Staubli VAL3: MoveTo.pgx

program MoveTo(pointRx x_pPoint, tool x_tTool, mdesc x_mDesc, num x_nMoveType, bool& x_bUnReachable)
  local string l_sMessage
  local joint l_jJoint
begin
  if pointToJoint(x_tTool,herej(),x_pPoint,l_jJoint)
    switch x_nMoveType
      case 0
        movel(x_pPoint,x_tTool,x_mDesc)
      break
      case 1
        movej(x_pPoint,x_tTool,x_mDesc)
      break
    endSwitch
  else
     x_bUnReachable=true
  endIf
end
